(* concatenate 4 strings *)
FUNCTION F_CONCAT4 : T_MaxString
VAR_INPUT
	strString1		: T_MaxString;
	strString2		: T_MaxString;
	strString3		: T_MaxString;
	strString4		: T_MaxString;
END_VAR
VAR
END_VAR
(*
-------------------------------------------------------------------------------------------------
Date		Version	Author	Comments
-------------------------------------------------------------------------------------------------
30/01/2015	3.00.00	PB		No change

-------------------------------------------------------------------------------------------------
05/02/2010	1.00.00	PB		Initial release

-------------------------------------------------------------------------------------------------
*)

F_CONCAT4 := CONCAT(strString1, strString2);
F_CONCAT4 := CONCAT(F_CONCAT4, strString3);
F_CONCAT4 := CONCAT(F_CONCAT4, strString4);

END_FUNCTION

(* stored: Version 1.1.0.1
   POU F_CONCAT4: Id {6440f64a-440b-4eee-bb7d-f50c988a6a7c}, SpecialFunc None *)
